{attribute 'linkalways'} 
{attribute 'no_explicit_call' := 'This FB is a CLASS and must be accessed using methods or properties'}
{attribute 'enable_dynamic_creation'}
FUNCTION_BLOCK Node_F_VN_DrawLineExp_TcVnVector4_LREAL EXTENDS VisionNode
VAR
    aLine : _TcVnVector4_LREAL;
    ipDestImage : _ITcVnImage;
    aColor : _TcVnVector4_LREAL;
    nThickness : _DINT(1);
    eLineType : _ETcVnLineType(ETcVnLineType.TCVN_LT_4_CONNECTED);
    nShift : _UDINT(0);
    hrPrev : _HRESULT(S_OK);
	hresult : _HRESULT(S_OK);
END_VAR

METHOD PUBLIC  Clone : I_Node
VAR
	pNode : POINTER TO Node_F_VN_DrawLineExp_TcVnVector4_LREAL;
END_VAR
pNode := __NEW(Node_F_VN_DrawLineExp_TcVnVector4_LREAL);
Clone := pNode^;
END_METHOD

METHOD FB_init : BOOL
VAR_INPUT
	bInitRetains : BOOL; // if TRUE, the retain variables are initialized (warm start / cold start)
	bInCopyCode : BOOL;  // if TRUE, the instance afterwards gets moved into the copy code (online change)
END_VAR
AddInput('aLine', aLine);
AddInput('ipDestImage', ipDestImage);
AddInput('aColor', aColor);
AddParameter('nThickness', nThickness);
AddParameter('eLineType', eLineType);
AddParameter('nShift', nShift);
AddInput('hrPrev', hrPrev);
AddOutput('ipDestImage', ipDestImage);
AddOutput('hresult',hresult);
END_METHOD

METHOD PROTECTED OnExecute
hresult.Value := F_VN_DrawLineExp_TcVnVector4_LREAL(
    aLine := aLine.Value,
	ipDestImage := ipDestImage.Value,
    aColor := aColor.Value,
    nThickness := nThickness.Value,
    eLineType := eLineType.Value,
    nShift := nShift.Value,
	hrPrev:= hrPrev.Value);
END_METHOD

METHOD PUBLIC PreExecutionCheck
VAR_INPUT
	Check : I_PreExecutionChecks;
END_VAR
Check.IsTrue(ipDestImage.IsValid, 'ipDestImage must contain an image');
Check.IsTrue(nThickness.Value >= 1, 'nThickness must be greater than or equal to 1');
END_METHOD

END_FUNCTION_BLOCK

(* stored: Version 1.1.0.1, ProductVersion 3.1.4024.15
   POU Node_F_VN_DrawLineExp_TcVnVector4_LREAL: Id {49e8e532-e2c5-4ad5-8c25-2b57f8e4a1e3}, SpecialFunc None
   Folder Constructor: Id {67608834-2017-4483-a519-552fc4a2302d}
   Method Clone: Id {aec67468-9356-42e2-8208-faad9479ac72}
   Method FB_init: Id {582b9c71-30ca-4b5b-a150-7ea7b3e1d9f9}
   Method OnExecute: Id {f5df553c-fd99-4266-b437-2cd88a03d229}
   Method PreExecutionCheck: Id {84c7ec7b-0c0c-471d-8a26-e93dde61c978} *)
